TYPE "Positioning_DOL_Machine_Wng"
VERSION : 0.1
// Block: Positioning_DOL_Machine_Wng
   STRUCT
      NotAutReady : Bool;
      MissingCnd_Minus : Bool;
      MissingCnd_Plus : Bool;
      Ax_NotHomed : Bool;
      Ax : OOAx_Wng;
      S120 : Struct
         Drive : Bool;
      END_STRUCT;
   END_STRUCT;

END_TYPE
